// Mitsubishi GX Works2 project: 램프5   PLC: Q02/Q02H

PROGRAM MAIN
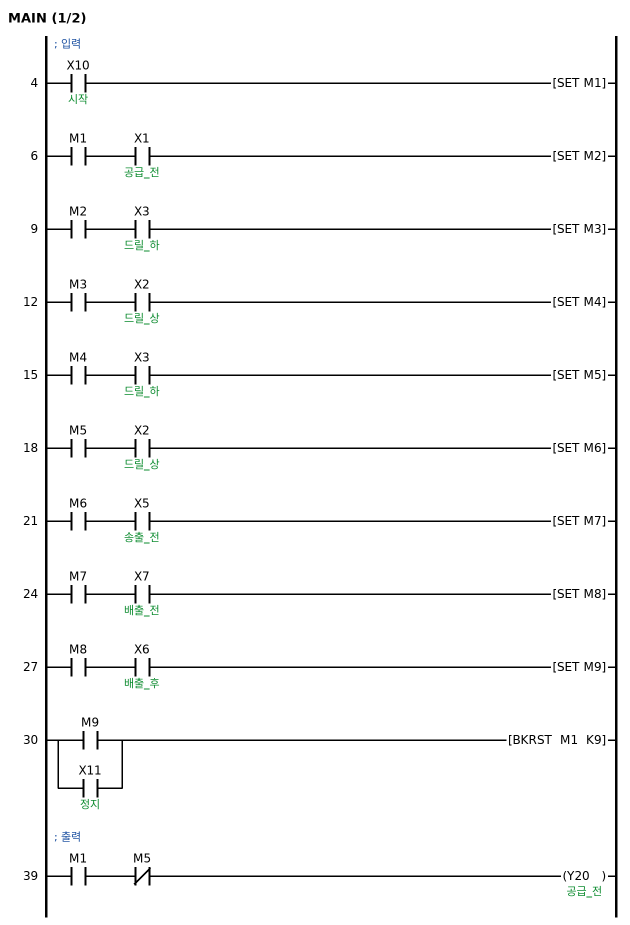
; 입력
4     LD      X10  ; 시작
      SET     M1
6     LD      M1
      AND     X1  ; 공급_전
      SET     M2
9     LD      M2
      AND     X3  ; 드릴_하
      SET     M3
12    LD      M3
      AND     X2  ; 드릴_상
      SET     M4
15    LD      M4
      AND     X3  ; 드릴_하
      SET     M5
18    LD      M5
      AND     X2  ; 드릴_상
      SET     M6
21    LD      M6
      AND     X5  ; 송출_전
      SET     M7
24    LD      M7
      AND     X7  ; 배출_전
      SET     M8
27    LD      M8
      AND     X6  ; 배출_후
      SET     M9
30    LD      M9
      OR      X11  ; 정지
      BKRST   M1 K9
; 출력
39    LD      M1
      ANI     M5
      OUT     Y20  ; 공급_전
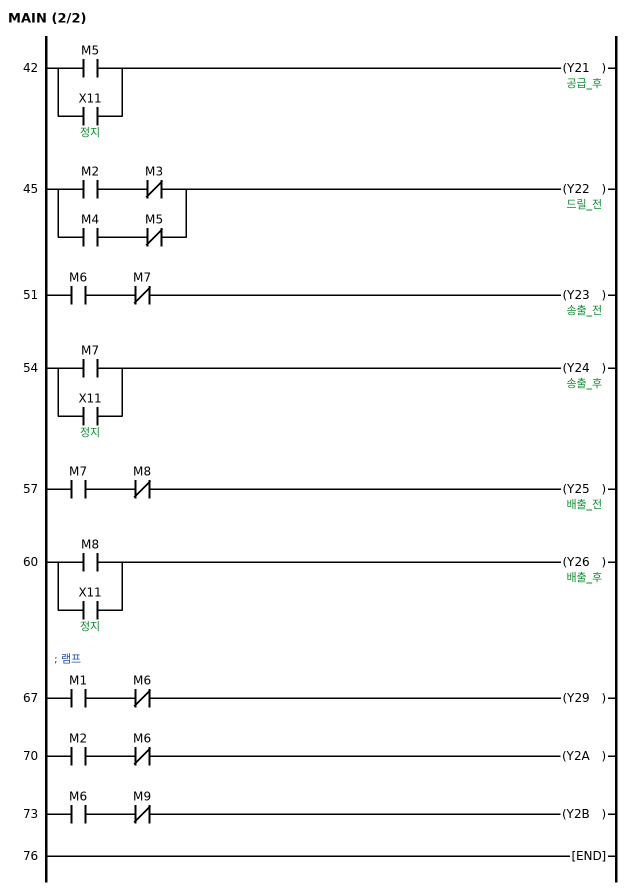
42    LD      M5
      OR      X11  ; 정지
      OUT     Y21  ; 공급_후
45    LD      M2
      ANI     M3
      LD      M4
      ANI     M5
      ORB
      OUT     Y22  ; 드릴_전
51    LD      M6
      ANI     M7
      OUT     Y23  ; 송출_전
54    LD      M7
      OR      X11  ; 정지
      OUT     Y24  ; 송출_후
57    LD      M7
      ANI     M8
      OUT     Y25  ; 배출_전
60    LD      M8
      OR      X11  ; 정지
      OUT     Y26  ; 배출_후
; 램프
67    LD      M1
      ANI     M6
      OUT     Y29
70    LD      M2
      ANI     M6
      OUT     Y2A
73    LD      M6
      ANI     M9
      OUT     Y2B
76    END
END_PROGRAM

// device comments not shown above
X0  ; 공급_후
X4  ; 송출_후
